{attribute 'GeneratedUsingTerminal: ER5151-0002-0018'}
{attribute addProperty BoxType "ER5151-0002-0018"}
{attribute addProperty Id "ENC_Status_compactAT %I*ENC_Status_compact_7D3464F320ENC_Control_compactAT %Q*ENC_Control_compact_21E2D14D6WcStateAT %I*WcState_9091E0EB2InfoDataAT %I*InfoData_94A18F5E2"}
{attribute addProperty CRC "3518367626"}
{attribute addProperty Size "30"}
TYPE ER5151_D1B6078A EXTENDS EtcSlaveTerminalBase_947E5A46 :
STRUCT
	{attribute addProperty Name "ENC_Status_compact"}
	ENC_Status_compact : ENC_Status_compact_7D3464F3;
	{attribute addProperty Name "ENC_Control_compact"}
	ENC_Control_compact : ENC_Control_compact_21E2D14D;
	{attribute addProperty Name "WcState"}
	WcState : WcState_9091E0EB;
	{attribute addProperty Name "InfoData"}
	InfoData : InfoData_94A18F5E;
END_STRUCT
END_TYPE

(* stored: Version 1.2.0.0, ProductVersion 3.1.4024.9
   DUT ER5151_D1B6078A: Id {0453192e-e995-49b7-990b-b5af09c4904a} *)
